Fanuc KAREL source: kd00074.KL

-- PROVISIONAL review KL for V1013-1; original PC SHA256 3d15144c25b13f4d601c8adca61408e93db9a6d14ba650d53437b438d921fa16
-- Incomplete behavior may be omitted. Consult companion uncertainty JSON. Do not deploy.
PROGRAM KD00074
%NOLOCKGROUP
VAR
  I : INTEGER
  J : INTEGER
  B : BOOLEAN
  R : REAL
  S : STRING[80]
BEGIN
  -- UNRESOLVED_PC offsets 5-7; opcodes 9C,3B
  -- UNRESOLVED_PC offsets 12-16; opcodes 7F
END KD00074
